(* IEC 61131-3 sources: CodesysTest/export/Function Blocks/SolenoidValves/FB_DoubleSolenoidClosedCenterActuator.pou/RetractAsserted.prop, 1 file *)

(* ---- Get.pm.st ---- *)
(*#-#-#-#-#-#-#-#-#-#---Declaration---#-#-#-#-#-#-#-#-#-#-#-#-#*)

VAR
END_VAR
(*#-#-#-#-#-#-#-#-#-#---Implementation---#-#-#-#-#-#-#-#-#-#-#-#-#*)

RetractAsserted := solenoid1 AND NOT solenoid0;
